FUNCTION_BLOCK FT_PIWL (* PI Controller with Anti-Windup *)
  (* Standard: 61499-1; Description: version 1.3	11. mar. 2009 programmer 	hugo tested by		oscat FT_PIWL is a PI controller. The PID controller works according to the fomula Y = IN *(KP+ KI * INTEG(e) ). a rst will reset the integrator to 0 lim_h and Lim_l set the possible output range of the controller. the output flag lim will signal that the output limits are active. the integrator ist equipped with anti wind-up circuitry which limits trhe total output ranke to lim_l and lim_h default values for KP = 1, KI = 1, ILIM_L = -1E37, iLIM_H = +1E38. *)
  (* Version 1.0, 2025-12-19, Coding-Assistent, initial API and implementation and/or initial documentation *)
  PACKAGE OSCAT::Basic::POUs::Engineering::Control;
  IMPORT eclipse4diac::core::TypeHash;
  IMPORT OSCAT::Basic::POUs::Engineering::measurements::T_PLC_US;
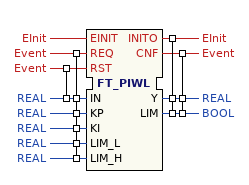
  EVENT_INPUT
    EINIT : EInit; (* Init Request *)
    REQ WITH IN, KP, KI, LIM_L, LIM_H; (* Normal Execution Request *)
    RST WITH IN; (* Reset Integrator *)
  END_EVENT
  EVENT_OUTPUT
    INITO : EInit WITH Y, LIM; (* Init Confirmation *)
    CNF WITH Y, LIM; (* Execution Confirmation *)
  END_EVENT
  VAR_INPUT
    IN : REAL; (* Process Variable / Error Input *)
    KP : REAL := 1.0; (* Proportional Gain *)
    KI : REAL := 1.0; (* Integral Gain *)
    LIM_L : REAL := -1.0E38; (* Lower Limit *)
    LIM_H : REAL := 1.0E38; (* Upper Limit *)
  END_VAR
  VAR_OUTPUT
    Y : REAL; (* Controller Output *)
    LIM : BOOL; (* Limit Reached Flag *)
  END_VAR
  VAR
    init : BOOL; (* Initialization Flag *)
    tx : UDINT; (* Current Time *)
    tc : REAL; (* Cycle Time (us) *)
    t_last : UDINT; (* Last Cycle Time *)
    in_last : REAL; (* Last Input Value *)
    i : REAL; (* Integrator Value *)
    p : REAL; (* Proportional Value *)
  END_VAR
  EC_STATES
    EINIT : EINIT -> INITO;
    REQ : REQ -> CNF;
    RST : RST -> CNF;
  END_STATES
  ALGORITHM EINIT IN ST:
(* Reset internal states *)
init := FALSE;
in_last := IN;
t_last := T_PLC_US();
i := 0.0;
tc := 0.0;
  END_ALGORITHM
  ALGORITHM RST IN ST:
this.EINIT();
init := TRUE;
  END_ALGORITHM
  ALGORITHM REQ IN ST:
(* initialize at power_up *)
IF NOT init THEN
	this.RST();
ELSE
	(* read last cycle time in Microseconds *)
	tx := T_PLC_US();
	tc := UDINT_TO_REAL(tx - t_last);
	t_last := tx;

		(* calculate proportional part *)
	p := KP * IN;

		(* run integrator *)
	i := (IN + in_last) * 5.0E-7 * KI * tc + i;
	in_last := IN;

		(* calculate output Y *)
	Y := p + i;

		(* check output for limits *)
	IF Y >= LIM_H THEN
		Y := LIM_H;
		IF KI <> 0.0 THEN
			i := LIM_H - p;
		ELSE
			i := 0.0;
		END_IF;
		LIM := TRUE;
	ELSIF Y <= LIM_L THEN
		Y := LIM_L;
		IF KI <> 0.0 THEN
			i := LIM_L - p;
		ELSE
			i := 0.0;
		END_IF;
		LIM := TRUE;
	ELSE
		LIM := FALSE;
	END_IF;
END_IF;
  END_ALGORITHM
END_FUNCTION_BLOCK
